// Library/Enumerations/Mode/ProcessingMode
{attribute 'qualified_only'}
// ------------------------------------------------------------------------- 
//  SRCI Robot Library                                                
// ------------------------------------------------------------------------- 
//                                                                           
//  Object:      ProcessingMode                                       
//  Author:      Thorsten Brach                                                
//  Date:        2024-06-01
//
//  Description:                                              
//   
//                                                                           
//  Copyright: 
//    (C) 2024 Thorsten Brach. All rights reserved                                                                                                                                            
//             Licensed under the LGPL-3.0 license.
//                                                                           
//  Disclaimer:                                                                           
//    This project is provided without any guarantee and can be used for   
//    private and commercial purposes. Any use is at the user’s 
//    own risk and responsibility.
//
// -------------------------------------------------------------------------
TYPE ProcessingMode :
(
  /// Command is buffered in sequence buffer and executed once
  BUFFERED := 0,
  /// Command is buffered in sequence buffer, aborts and empties previous commands in sequence buffer, and is executed once
  ABORTING := 1,
  /// Command is buffered in parallel buffer and executed once
  PARALLEL := 2,
  /// Command is buffered in parallel buffer and executed repeatedly until deliberate deactivation by user
  CONTINUOUS := 3,
  /// CMD execution is stopped and/or CMD is removed from the buffer
  DEACTIVATE := 9,
  /// Command is buffered in sequence buffer and executed once (Trigger based)
  TRIGGER_BUFFERED := 10,
  /// Command is buffered in sequence buffer, aborts and empties previous commands in sequence buffer, and is executed once (Trigger based)
  TRIGGER_ABORTING := 11,
  /// Command is buffered in parallel buffer and executed once (Trigger based)
  TRIGGER_ONCE := 12,
  /// Command is buffered in parallel buffer and executed repeatedly until deliberate deactivation by user (Trigger based)
  TRIGGER_CONTINUOUS := 13,
  /// Command is buffered and executed multiple times when triggered. The CMD remains in the buffer until removed by the user.
  TRIGGER_MULTIPLE := 14
)USINT;
END_TYPE

// Library/Enumerations/Mode/ResistanceForceMode
{attribute 'qualified_only'}
// ------------------------------------------------------------------------- 
//  SRCI Robot Library                                                
// ------------------------------------------------------------------------- 
//                                                                           
//  Object:      ResistanceForceMode                                       
//  Author:      Thorsten Brach                                                
//  Date:        2024-06-01
//
//  Description:                                              
//   
//                                                                           
//  Copyright: 
//    (C) 2024 Thorsten Brach. All rights reserved                                                                                                                                            
//             Licensed under the LGPL-3.0 license.
//                                                                           
//  Disclaimer:                                                                           
//    This project is provided without any guarantee and can be used for   
//    private and commercial purposes. Any use is at the user’s 
//    own risk and responsibility.
//
// -------------------------------------------------------------------------
TYPE ResistanceForceMode :
(
  /// 0 (default): ResistanceForceTCP.
  /// Set "0" to set the resistance of the RA against the external force at the TCP.
  RESISTANCE_FORCE_TCP := 0,
  
  /// 1: ResistanceForceAxis.
  /// Set "1" to set the resistance of the RA against the external force for each axis independently.
  RESISTANCE_FORCE_AXIS := 1
)USINT;
END_TYPE

// Library/Enumerations/Mode/ReturnMode
{attribute 'qualified_only'}
TYPE ReturnMode :
(
  /// Interrupt position
  INTERRUPT_POSITION := 0,
  /// End position
  END_POSITION := 1
)BYTE;
END_TYPE

// Library/Enumerations/Mode/SensorConnectionMode
{attribute 'qualified_only'}
// ------------------------------------------------------------------------- 
//  SRCI Robot Library                                                
// ------------------------------------------------------------------------- 
//                                                                           
//  Object:      SensorConnectionMode                                       
//  Author:      Thorsten Brach                                                
//  Date:        2024-06-01
//
//  Description:                                              
//   
//                                                                           
//  Copyright: 
//    (C) 2024 Thorsten Brach. All rights reserved                                                                                                                                            
//             Licensed under the LGPL-3.0 license.
//                                                                           
//  Disclaimer:                                                                           
//    This project is provided without any guarantee and can be used for   
//    private and commercial purposes. Any use is at the user’s 
//    own risk and responsibility.
//
// -------------------------------------------------------------------------
TYPE SensorConnectionMode :
(
  /// RC sensor and algorithm
  /// Force-Torque-Sensor connected to RC
  /// Control algorithm in RC
  RC_SENSOR_ALGORITHM := 0,
  
  /// PLC sensor and RC algorithm
  /// Force-Torque-Sensor connected to PLC
  /// Control algorithm in RC
  PLC_SENSOR_RC_ALGORITHM := 1,
  
  /// PLC sensor and algorithm
  /// Force-Torque-Sensor connected to PLC
  /// Control algorithm in PLC
  PLC_SENSOR_ALGORITHM := 2
)USINT;
END_TYPE

// Library/Enumerations/Mode/SingularityAvoidanceMode
{attribute 'qualified_only'}
// ------------------------------------------------------------------------- 
//  SRCI Robot Library                                                
// ------------------------------------------------------------------------- 
//                                                                           
//  Object:      SingularityAvoidanceMode                                       
//  Author:      Thorsten Brach                                                
//  Date:        2024-06-01
//
//  Description:                                              
//   
//                                                                           
//  Copyright: 
//    (C) 2024 Thorsten Brach. All rights reserved                                                                                                                                            
//             Licensed under the LGPL-3.0 license.
//                                                                           
//  Disclaimer:                                                                           
//    This project is provided without any guarantee and can be used for   
//    private and commercial purposes. Any use is at the user’s 
//    own risk and responsibility.
//
// -------------------------------------------------------------------------
TYPE SingularityAvoidanceMode :
(
  /// 0: NoChange (default)
  /// Allow movement of one or more joints to avoid singularities without a change of the orientation
  NO_CHANGE := 0,
  
  /// 1: Lock J4
  /// Lock the 4th joint to avoid singularities
  LOCK_J4 := 1,
  
  /// 2: ToolOrientation
  /// Allow a small movement of the tool orientation to avoid singularities
  TOOL_ORIENTATION := 2
)USINT;
END_TYPE

// Library/Enumerations/Mode/SplineMode
{attribute 'qualified_only'}
// ------------------------------------------------------------------------- 
//  SRCI Robot Library                                                
// ------------------------------------------------------------------------- 
//                                                                           
//  Object:      SplineMode                                       
//  Author:      Thorsten Brach                                                
//  Date:        2024-06-01
//
//  Description:                                              
//   
//                                                                           
//  Copyright: 
//    (C) 2024 Thorsten Brach. All rights reserved                                                                                                                                            
//             Licensed under the LGPL-3.0 license.
//                                                                           
//  Disclaimer:                                                                           
//    This project is provided without any guarantee and can be used for   
//    private and commercial purposes. Any use is at the user’s 
//    own risk and responsibility.
//
// -------------------------------------------------------------------------
TYPE SplineMode :
(
  /// 0: Discrete Points
  DISCRETE_POINTS := 0,
  /// 1: Bézier Spline
  BEZIER_SPLINE := 1,
  /// 2: B-Splines
  B_SPLINES := 2,
  /// 3: Cubic Hermite Spline
  CUBIC_HERMITE_SPLINE := 3,
  /// 4: C-Splines
  C_SPLINES := 4
)UINT;
END_TYPE

// Library/Enumerations/Mode/StepMode
{attribute 'qualified_only'}
// ------------------------------------------------------------------------- 
//  SRCI Robot Library                                                
// ------------------------------------------------------------------------- 
//                                                                           
//  Object:      StepMode                                       
//  Author:      Thorsten Brach                                                
//  Date:        2024-06-01
//
//  Description:                                              
//   
//                                                                           
//  Copyright: 
//    (C) 2024 Thorsten Brach. All rights reserved                                                                                                                                            
//             Licensed under the LGPL-3.0 license.
//                                                                           
//  Disclaimer:                                                                           
//    This project is provided without any guarantee and can be used for   
//    private and commercial purposes. Any use is at the user’s 
//    own risk and responsibility.
//
// -------------------------------------------------------------------------
TYPE StepMode :
(
  /// StepMode is deactivated
  DEACTIVATE := 0,
  /// Blending
  /// • The robot moves on the blended trajectory
  /// • The movement is interrupted when the active segment changes
  BLENDING := 1,
  ///Exact stop
  /// • The robot moves to the defined target positions without blending
  /// • The movement is interrupted when the defined target position is reached
  EXACT_STOP := 2
)USINT;
END_TYPE

// Library/Enumerations/Mode/StopMode
{attribute 'qualified_only'}
// ------------------------------------------------------------------------- 
//  SRCI Robot Library                                                
// ------------------------------------------------------------------------- 
//                                                                           
//  Object:      StopMode                                       
//  Author:      Thorsten Brach                                                
//  Date:        2024-06-01
//
//  Description:                                              
//   
//                                                                           
//  Copyright: 
//    (C) 2024 Thorsten Brach. All rights reserved                                                                                                                                            
//             Licensed under the LGPL-3.0 license.
//                                                                           
//  Disclaimer:                                                                           
//    This project is provided without any guarantee and can be used for   
//    private and commercial purposes. Any use is at the user’s 
//    own risk and responsibility.
//
// -------------------------------------------------------------------------
TYPE StopMode :
(
  /// 0: Stop via JobID (default)
  /// TargetID is interpreted as JobID
  /// All instances of the defined JobID are stopped
  STOP_JOB_ID := 0,  
  /// 1: Stop via InstanceID
  /// TargetID is interpreted as InstanceID
  /// The instance of the defined InstanceID is stopped
  STOP_INSTANCE_ID := 1,  
  /// 2: Stop all subprograms
  /// All subprograms independent of the input parameter value of TargetID are stopped
  STOP_ALL_SUBPROGRAMS := 2
)USINT;
END_TYPE

// Library/Enumerations/Mode/SyncInMode
{attribute 'qualified_only'}
// ------------------------------------------------------------------------- 
//  SRCI Robot Library                                                
// ------------------------------------------------------------------------- 
//                                                                           
//  Object:      SyncInMode                                       
//  Author:      Thorsten Brach                                                
//  Date:        2024-06-01
//
//  Description:                                              
//   
//                                                                           
//  Copyright: 
//    (C) 2024 Thorsten Brach. All rights reserved                                                                                                                                            
//             Licensed under the LGPL-3.0 license.
//                                                                           
//  Disclaimer:                                                                           
//    This project is provided without any guarantee and can be used for   
//    private and commercial purposes. Any use is at the user’s 
//    own risk and responsibility.
//
// -------------------------------------------------------------------------
TYPE SyncInMode :
(
  /// • When work piece enters "SyncInZone"
  /// • Start synchronization as soon as possible within defined acceleration and velocity limits
  IN_SYNC_IN_ZONE := 0,
  /// • Start synchronization after specific distance after execution
  /// • "SynInZone" ignored
  AFTER_DISTANCE := 1,
  /// • Start synchronization after specific time after execution
  /// • "SynInZone" ignored
  AFTER_TIME := 2,
  /// • As soon as possible within defined acceleration and velocity limits
  /// • "SynInZone" ignored
  IMMEDIATELY := 3
)USINT;
END_TYPE

// Library/Enumerations/Mode/SyncMode
{attribute 'qualified_only'}
// ------------------------------------------------------------------------- 
//  SRCI Robot Library                                                
// ------------------------------------------------------------------------- 
//                                                                           
//  Object:      SyncMode                                       
//  Author:      Thorsten Brach                                                
//  Date:        2024-06-01
//
//  Description:                                              
//   
//                                                                           
//  Copyright: 
//    (C) 2024 Thorsten Brach. All rights reserved                                                                                                                                            
//             Licensed under the LGPL-3.0 license.
//                                                                           
//  Disclaimer:                                                                           
//    This project is provided without any guarantee and can be used for   
//    private and commercial purposes. Any use is at the user’s 
//    own risk and responsibility.
//
// -------------------------------------------------------------------------
TYPE SyncMode :
(
  /// No synchronization will be executed
  NO_SYNCHRONIZATION := 0,
  /// Server data will be overwritten immediately by client data
  CLIENT_TO_SERVER := 1,
  /// Client data will be overwritten immediately by server data
  SERVER_TO_CLIENT := 2,
  /// Server or client data will be overwritten immediately by changed data
  AUTOMATIC := 3
)USINT;
END_TYPE

// Library/Enumerations/Mode/ThresholdMode
{attribute 'qualified_only'}
// ------------------------------------------------------------------------- 
//  SRCI Robot Library                                                
// ------------------------------------------------------------------------- 
//                                                                           
//  Object:      ThresholdMode                                       
//  Author:      Thorsten Brach                                                
//  Date:        2024-06-01
//
//  Description:                                              
//   
//                                                                           
//  Copyright: 
//    (C) 2024 Thorsten Brach. All rights reserved                                                                                                                                            
//             Licensed under the LGPL-3.0 license.
//                                                                           
//  Disclaimer:                                                                           
//    This project is provided without any guarantee and can be used for   
//    private and commercial purposes. Any use is at the user’s 
//    own risk and responsibility.
//
// -------------------------------------------------------------------------
TYPE ThresholdMode :
(
  /// Automatic.
  AUTOMATIC := 0,
  /// Manual (according to LimitAxis)
  MANUAL    := 1
)USINT;
END_TYPE

// Library/Enumerations/Mode/ToolCalculationMode
{attribute 'qualified_only'}
// ------------------------------------------------------------------------- 
//  SRCI Robot Library                                                
// ------------------------------------------------------------------------- 
//                                                                           
//  Object:      ToolCalculationMode                                       
//  Author:      Thorsten Brach                                                
//  Date:        2024-06-01
//
//  Description:                                              
//   
//                                                                           
//  Copyright: 
//    (C) 2024 Thorsten Brach. All rights reserved                                                                                                                                            
//             Licensed under the LGPL-3.0 license.
//                                                                           
//  Disclaimer:                                                                           
//    This project is provided without any guarantee and can be used for   
//    private and commercial purposes. Any use is at the user’s 
//    own risk and responsibility.
//
// -------------------------------------------------------------------------
TYPE ToolCalculationMode :
(
  /// 0: Two Point + Z-Method (default)
  TWO_POINT_Z_METHOD := 0,        
  /// 1: Three-Point-Method
  THREE_POINT_METHOD := 1,        
  /// 2: Four-Point-Method
  FOUR_POINT_METHOD := 2,        
  /// 3: Five-Point-Method
  FIVE_POINT_METHOD := 3,        
  /// 4: Six-Point-Method
  SIX_POINT_METHOD := 4,        
  /// 5: ABC-World-Method
  ABC_WORLD_METHOD := 5,        
  /// 6: ABC-Two-Point-Method
  ABC_TWO_POINT_METHOD := 6
)SINT;
END_TYPE

// Library/Enumerations/Mode/TrajectoryMode
{attribute 'qualified_only'}
// ------------------------------------------------------------------------- 
//  SRCI Robot Library                                                
// ------------------------------------------------------------------------- 
//                                                                           
//  Object:      TrajectoryMode                                       
//  Author:      Thorsten Brach                                                
//  Date:        2024-06-01
//
//  Description:                                              
//   
//                                                                           
//  Copyright: 
//    (C) 2024 Thorsten Brach. All rights reserved                                                                                                                                            
//             Licensed under the LGPL-3.0 license.
//                                                                           
//  Disclaimer:                                                                           
//    This project is provided without any guarantee and can be used for   
//    private and commercial purposes. Any use is at the user’s 
//    own risk and responsibility.
//
// -------------------------------------------------------------------------
TYPE TrajectoryMode :
(
  /// Invalid (default)
  INVALID := 0,
  /// Linear movement
  LINEAR_MOVEMENT := 1,
  /// PTP movement
  PTP_MOVEMENT := 2
)USINT;
END_TYPE

// Library/Enumerations/Mode/TransformMode
{attribute 'qualified_only'}
// ------------------------------------------------------------------------- 
//  SRCI Robot Library                                                
// ------------------------------------------------------------------------- 
//                                                                           
//  Object:      TransformMode                                       
//  Author:      Thorsten Brach                                                
//  Date:        2024-06-01
//
//  Description:                                              
//   
//                                                                           
//  Copyright: 
//    (C) 2024 Thorsten Brach. All rights reserved                                                                                                                                            
//             Licensed under the LGPL-3.0 license.
//                                                                           
//  Disclaimer:                                                                           
//    This project is provided without any guarantee and can be used for   
//    private and commercial purposes. Any use is at the user’s 
//    own risk and responsibility.
//
// -------------------------------------------------------------------------
TYPE TransformMode :
(
  /// 0 (default): Mirror at Point with mirroring of the target position’s orientation
  /// Requires for the mirror Point the "TransformationParameter_1" and the "TransformationParameter_2" set to "Not used"
  MIRROR_AT_POINT := 0,  
  /// 1: Mirror at Straight Line with mirroring of the target position’s orientation
  /// Requires for the Straight Line the "TransformationParameter_1" and the "TransformationParameter_2" set to "X-Axis", "Y-Axis" or "Z-Axis"
  MIRROR_AT_STRAIGHT_LINE := 1,  
  /// 2: Mirror at Plane with mirroring of the target position’s orientation
  /// Requires for the Plane the "TransformationParameter_1" and the "TransformationParameter_2" set to "XY-Axis", "XZ-Axis" or "YZ-Axis"
  MIRROR_AT_PLANE := 2,  
  /// 3: Rotate around Straight Line with rotation of the target position’s orientation
  /// Requires for the Straight Line the "TransformationParameter_1" and the "TransformationParameter_2" set to "X-Axis", "Y-Axis" or "Z-Axis"
  /// Requires for the parameter "RotationAngle"
  ROTATE_AROUND_STRAIGHT_LINE := 3,  
  /// 4: Shift by Vector
  /// Requires for the shifting Vector defined by the Point the "TransformationParameter_1" and the "TransformationParameter_2" set to "Not used"
  /// Requires for the shifting shortest Vector to the Straight Line the "TransformationParameter_1" and the "TransformationParameter_2" set to "X-Axis", "Y-Axis" or "Z-Axis"
  /// Requires for the shifting shortest Vector to the Plane the "TransformationParameter_1" and the "TransformationParameter_2" set to "XY-Axis", "XZ-Axis" or "YZ-Axis"
  SHIFT_BY_VECTOR := 4
)SINT;
END_TYPE

// Library/Enumerations/Mode/TriggerModeIo
{attribute 'qualified_only'}
// ------------------------------------------------------------------------- 
//  SRCI Robot Library                                                
// ------------------------------------------------------------------------- 
//                                                                           
//  Object:      TriggerModeIo                                       
//  Author:      Thorsten Brach                                                
//  Date:        2024-06-01
//
//  Description:                                              
//   
//                                                                           
//  Copyright: 
//    C) 2024 Thorsten Brach. All rights reserved                                                                                                                                            
//             Licensed under the LGPL-3.0 license.
//                                                                           
//  Disclaimer:                                                                           
//    This project is provided without any guarantee and can be used for   
//    private and commercial purposes. Any use is at the user’s 
//    own risk and responsibility.
//
// -------------------------------------------------------------------------
TYPE TriggerModeIo :
(
  /// Invalid (default)
  INVALID := 0,  
  /// Digital Input Rising Edge
  DIGITAL_INPUT_RISING_EDGE := 10,
  /// Digital Input Falling Edge
  DIGITAL_INPUT_FALLING_EDGE := 11,
  /// Digital Input Rising or Falling Edge
  DIGITAL_INPUT_RISING_OR_FALLING_EDGE := 12,
  /// Digital Input Rising or Falling Edge (Inverted)
  DIGITAL_INPUT_RISING_OR_FALLING_EDGE_INVERTED := 13,
  /// Digital Output Rising Edge
  DIGITAL_OUTPUT_RISING_EDGE := 20,
  /// Digital Output Falling Edge
  DIGITAL_OUTPUT_FALLING_EDGE := 21,
  /// Digital Output Rising or Falling Edge
  DIGITAL_OUTPUT_RISING_OR_FALLING_EDGE := 22,
  /// Digital Output Rising or Falling Edge (Inverted)
  DIGITAL_OUTPUT_RISING_OR_FALLING_EDGE_INVERTED := 23,
  /// Analog Input Exceeding Defined Threshold
  ANALOG_INPUT_EXCEEDING_DEFINED_THRESHOLD := 30,
  /// Analog Input Falling Below Defined Threshold
  ANALOG_INPUT_FALLING_BELOW_DEFINED_THRESHOLD := 31,
  /// Analog Input Exceeding or Falling Below Defined Threshold
  ANALOG_INPUT_EXCEEDING_OR_FALLING_BELOW_DEFINED_THRESHOLD := 32,
  /// Analog Input Exceeding or Falling Below Defined Threshold (Inverted)
  ANALOG_INPUT_EXCEEDING_OR_FALLING_BELOW_DEFINED_THRESHOLD_INVERTED := 33,
  /// Analog Input Entering Defined Range
  ANALOG_INPUT_ENTERING_DEFINED_RANGE := 34,
  /// Analog Input Leaving Defined Range
  ANALOG_INPUT_LEAVING_DEFINED_RANGE := 35,
  /// Analog Input Entering or Leaving Defined Range
  ANALOG_INPUT_ENTERING_OR_LEAVING_DEFINED_RANGE := 36,
  /// Analog Input Entering or Leaving Defined Range (Inverted)
  ANALOG_INPUT_ENTERING_OR_LEAVING_DEFINED_RANGE_INVERTED := 37,
  /// Analog Output Exceeding Defined Threshold
  ANALOG_OUTPUT_EXCEEDING_DEFINED_THRESHOLD := 40,
  /// Analog Output Falling Below Defined Threshold
  ANALOG_OUTPUT_FALLING_BELOW_DEFINED_THRESHOLD := 41,
  /// Analog Output Exceeding or Falling Below Defined Threshold
  ANALOG_OUTPUT_EXCEEDING_OR_FALLING_BELOW_DEFINED_THRESHOLD := 42,
  /// Analog Output Exceeding or Falling Below Defined Threshold (Inverted)
  ANALOG_OUTPUT_EXCEEDING_OR_FALLING_BELOW_DEFINED_THRESHOLD_INVERTED := 43,
  /// Analog Output Entering Defined Range
  ANALOG_OUTPUT_ENTERING_DEFINED_RANGE := 44,
  /// Analog Output Leaving Defined Range
  ANALOG_OUTPUT_LEAVING_DEFINED_RANGE := 45,
  /// Analog Output Entering or Leaving Defined Range
  ANALOG_OUTPUT_ENTERING_OR_LEAVING_DEFINED_RANGE := 46,
  /// Analog Output Entering or Leaving Defined Range (Inverted)
  ANALOG_OUTPUT_ENTERING_OR_LEAVING_DEFINED_RANGE_INVERTED := 47,
  /// Integer Register Exceeding Defined Threshold
  INTEGER_REGISTER_EXCEEDING_DEFINED_THRESHOLD := 50,
  /// Integer Register Falling Below Defined Threshold
  INTEGER_REGISTER_FALLING_BELOW_DEFINED_THRESHOLD := 51,
  /// Integer Register Exceeding or Falling Below Defined Threshold
  INTEGER_REGISTER_EXCEEDING_OR_FALLING_BELOW_DEFINED_THRESHOLD := 52,
  /// Integer Register Exceeding or Falling Below Defined Value (Inverted)
  INTEGER_REGISTER_EXCEEDING_OR_FALLING_BELOW_DEFINED_VALUE_INVERTED := 53,
  /// Integer Register Entering Defined Range
  INTEGER_REGISTER_ENTERING_DEFINED_RANGE := 54,
  /// Integer Register Leaving Defined Range
  INTEGER_REGISTER_LEAVING_DEFINED_RANGE := 55,
  /// Integer Register Entering or Leaving Defined Range
  INTEGER_REGISTER_ENTERING_OR_LEAVING_DEFINED_RANGE := 56,
  /// Integer Register Entering or Leaving Defined Range (Inverted)
  INTEGER_REGISTER_ENTERING_OR_LEAVING_DEFINED_RANGE_INVERTED := 57,
  /// Real Register Exceeding Defined Threshold
  REAL_REGISTER_EXCEEDING_DEFINED_THRESHOLD := 60,
  /// Real Register Falling Below Defined Threshold
  REAL_REGISTER_FALLING_BELOW_DEFINED_THRESHOLD := 61,
  /// Real Register Exceeding or Falling Below Defined Threshold
  REAL_REGISTER_EXCEEDING_OR_FALLING_BELOW_DEFINED_THRESHOLD := 62,
  /// Real Register Exceeding or Falling Below Defined Threshold (Inverted)
  REAL_REGISTER_EXCEEDING_OR_FALLING_BELOW_DEFINED_THRESHOLD_INVERTED := 63,
  /// Real Register Entering Defined Range
  REAL_REGISTER_ENTERING_DEFINED_RANGE := 64,
  /// Real Register Leaving Defined Range
  REAL_REGISTER_LEAVING_DEFINED_RANGE := 65,
  /// Real Register Entering or Leaving Defined Range
  REAL_REGISTER_ENTERING_OR_LEAVING_DEFINED_RANGE := 66,
  /// Real Register Entering or Leaving Defined Range (Inverted)
  REAL_REGISTER_ENTERING_OR_LEAVING_DEFINED_RANGE_INVERTED := 67
)SINT;
END_TYPE

// Library/Enumerations/Mode/TriggerModeLimit
{attribute 'qualified_only'}
// ------------------------------------------------------------------------- 
//  SRCI Robot Library                                                
// ------------------------------------------------------------------------- 
//                                                                           
//  Object:      TriggerModeLimit                                       
//  Author:      Thorsten Brach                                                
//  Date:        2024-06-01
//
//  Description:                                              
//   
//                                                                           
//  Copyright: 
//    (C) 2024 Thorsten Brach. All rights reserved                                                                                                                                            
//             Licensed under the LGPL-3.0 license.
//                                                                           
//  Disclaimer:                                                                           
//    This project is provided without any guarantee and can be used for   
//    private and commercial purposes. Any use is at the user’s 
//    own risk and responsibility.
//
// -------------------------------------------------------------------------
TYPE TriggerModeLimit :
(
  /// 0: Invalid (default)
  INVALID := 0,
  /// 1: Joint current in mA
  JOINT_CURRENT := 1,
  /// 2: Force in Nm
  FORCE := 2,
  /// 3: Following error. The distance of the robot position from the path that was calculated
  FOLLOWING_ERROR := 3,
  /// Temperature in °C
  TEMPERATURE := 4  
)SINT;
END_TYPE

// Library/Enumerations/Mode/TriggerModeMeasurement
{attribute 'qualified_only'}
// ------------------------------------------------------------------------- 
//  SRCI Robot Library                                                
// ------------------------------------------------------------------------- 
//                                                                           
//  Object:      TriggerModeMeasurement                                       
//  Author:      Thorsten Brach                                                
//  Date:        2024-06-01
//
//  Description:                                              
//   
//                                                                           
//  Copyright: 
//    (C) 2024 Thorsten Brach. All rights reserved                                                                                                                                            
//             Licensed under the LGPL-3.0 license.
//                                                                           
//  Disclaimer:                                                                           
//    This project is provided without any guarantee and can be used for   
//    private and commercial purposes. Any use is at the user’s 
//    own risk and responsibility.
//
// -------------------------------------------------------------------------
TYPE TriggerModeMeasurement :
(
  /// (default) No trigger related behavior
  NO_TRIGGER := 0,
  /// 1: Starts the measurement with the positive trigger event and stops it with the negative trigger event 
  ///    when the trigger function with the identical EmitterID is activated.
  POSITIVE_START_NEGATIVE_STOP := 1,
  /// 2: Starts and stops the measurement with the positive trigger event 
  ///    when the trigger function with the identical EmitterID is activated.
  POSITIVE_START_STOP := 2
)USINT;
END_TYPE

// Library/Enumerations/Mode/TriggerReactionMode
{attribute 'qualified_only'}
// ------------------------------------------------------------------------- 
//  SRCI Robot Library                                                
// ------------------------------------------------------------------------- 
//                                                                           
//  Object:      TriggerReactionMode                                       
//  Author:      Thorsten Brach                                                
//  Date:        2024-06-01
//
//  Description:                                              
//   
//                                                                           
//  Copyright: 
//    (C) 2024 Thorsten Brach. All rights reserved                                                                                                                                            
//             Licensed under the LGPL-3.0 license.
//                                                                           
//  Disclaimer:                                                                           
//    This project is provided without any guarantee and can be used for   
//    private and commercial purposes. Any use is at the user’s 
//    own risk and responsibility.
//
// -------------------------------------------------------------------------
TYPE TriggerReactionMode :
(
/// No reaction (default).
  NO_REACTION := 0,
  /// Interrupt: Robot movement is paused. Movement can be continued by function GroupContinue.
  INTERRUPT := 1,
  /// GroupStop: Robot stops the movement and brings all axes to a halt. Movements aborted by this command cannot be continued.
  GROUP_STOP := 2,
  /// Disable robot: The robot’s drives are disabled. This leads to the robot state "Not enabled" (see chapter 5.5.3).
  DISABLE_ROBOT := 3,
  /// Stop actual motion command: Robot movement is paused. Movement can be continued by the next motion command.
  STOP_ACTUAL_MOTION_COMMAND := 4
)SINT;
END_TYPE

// Library/Enumerations/Mode/TurnMode
{attribute 'qualified_only'}
// ------------------------------------------------------------------------- 
//  SRCI Robot Library                                                
// ------------------------------------------------------------------------- 
//                                                                           
//  Object:      TurnMode                                       
//  Author:      Thorsten Brach                                                
//  Date:        2024-06-01
//
//  Description:                                              
//   
//                                                                           
//  Copyright: 
//    (C) 2024 Thorsten Brach. All rights reserved                                                                                                                                            
//             Licensed under the LGPL-3.0 license.
//                                                                           
//  Disclaimer:                                                                           
//    This project is provided without any guarantee and can be used for   
//    private and commercial purposes. Any use is at the user’s 
//    own risk and responsibility.
//
// -------------------------------------------------------------------------
TYPE TurnMode :
(
  /// Use TurnNumber in position
  USE_TURN_NUMBER := 0,
  ///  Do not change TurnNumber with this movement
  SAME            := 1,
  /// TurnNumber in position is not used but the Robot is free to change TurnNumber
  FREE            := 2
)USINT;
END_TYPE

// Library/Enumerations/Mode/WorkAreaReactionMode
{attribute 'qualified_only'}
// ------------------------------------------------------------------------- 
//  SRCI Robot Library                                                
// ------------------------------------------------------------------------- 
//                                                                           
//  Object:      WorkAreaReactionMode                                       
//  Author:      Thorsten Brach                                                
//  Date:        2024-06-01
//
//  Description:                                              
//   
//                                                                           
//  Copyright: 
//    (C) 2024 Thorsten Brach. All rights reserved                                                                                                                                            
//             Licensed under the LGPL-3.0 license.
//                                                                           
//  Disclaimer:                                                                           
//    This project is provided without any guarantee and can be used for   
//    private and commercial purposes. Any use is at the user’s 
//    own risk and responsibility.
//
// -------------------------------------------------------------------------
TYPE WorkAreaReactionMode :
(
  /// 0: No reaction (default)
  /// • RC reports violation
  /// • Robot is not stopped
  NO_REACTION := 0,
  /// 
  /// 1: Abort
  /// • RC reports violation
  /// • RC returns error
  /// • Robot is stopped
  /// • Sequence buffer emptied
  ABORT := 1,
  /// 2: Interrupt
  /// • RC reports violation
  /// • Robot movement is paused
  /// • Movement can be continued by function GroupContinue
   INTERRUPT := 2
)USINT;
END_TYPE

// Library/Enumerations/State/ActiveCommandRegisterState
{attribute 'qualified_only'}
// ------------------------------------------------------------------------- 
//  SRCI Robot Library                                                
// ------------------------------------------------------------------------- 
//                                                                           
//  Object:      ActiveCommandRegisterState                                       
//  Author:      Thorsten Brach                                                
//  Date:        2024-06-01
//
//  Description:                                              
//   
//                                                                           
//  Copyright: 
//    (C) 2024 Thorsten Brach. All rights reserved                                                                                                                                            
//             Licensed under the LGPL-3.0 license.
//                                                                           
//  Disclaimer:                                                                           
//    This project is provided without any guarantee and can be used for   
//    private and commercial purposes. Any use is at the user’s 
//    own risk and responsibility.
//
// -------------------------------------------------------------------------
TYPE ActiveCommandRegisterState :
(
  /// IS_FREE denotes not used but available resources (empty slots in the ACR).
  IS_FREE        := 0,
  /// IS_PROCESSING CMDs are actively being processed by client or server. 
  /// In terms of CMD category, IS_PROCESSING also describes commands whose tasks are not currently being executed (not ACTIVE), 
  /// but e.g. a CMD waiting in the Sequence buffer.
  IS_PROCESSING := 1,
  /// IS_FINAL states are reached on CMD termination. Execution of this Task has been finished and its results can be examined.
  IS_FINAL    := 2
);
END_TYPE

// Library/Enumerations/State/BufferStateCmd
{attribute 'qualified_only'}
// ------------------------------------------------------------------------- 
//  SRCI Robot Library                                                
// ------------------------------------------------------------------------- 
//                                                                           
//  Object:      BufferStateCmd                                       
//  Author:      Thorsten Brach                                                
//  Date:        2024-06-01
//
//  Description:                                              
//   
//                                                                           
//  Copyright: 
//    (C) 2024 Thorsten Brach. All rights reserved                                                                                                                                            
//             Licensed under the LGPL-3.0 license.
//                                                                           
//  Disclaimer:                                                                           
//    This project is provided without any guarantee and can be used for   
//    private and commercial purposes. Any use is at the user’s 
//    own risk and responsibility.
//
// -------------------------------------------------------------------------
TYPE BufferStateCmd :
(
 // PDF Page 353 
  EMPTY            := 0,
  CREATED          := 1,
  UPDATE_AVAILABLE := 2,
  SENDING          := 3,
  PROCESSED        := 4  
);
END_TYPE

// Library/Enumerations/State/BufferStateRsp
{attribute 'qualified_only'}
// ------------------------------------------------------------------------- 
//  SRCI Robot Library                                                
// ------------------------------------------------------------------------- 
//                                                                           
//  Object:      BufferStateRsp                                       
//  Author:      Thorsten Brach                                                
//  Date:        2024-06-01
//
//  Description:                                              
//   
//                                                                           
//  Copyright: 
//    (C) 2024 Thorsten Brach. All rights reserved                                                                                                                                            
//             Licensed under the LGPL-3.0 license.
//                                                                           
//  Disclaimer:                                                                           
//    This project is provided without any guarantee and can be used for   
//    private and commercial purposes. Any use is at the user’s 
//    own risk and responsibility.
//
// -------------------------------------------------------------------------
TYPE BufferStateRsp :
(
 // PDF Seite 353 
  EMPTY            := 0,
  RECEIVING        := 1,
  RECEIVED         := 2,
  PROCESSED        := 3  
);
END_TYPE

// Library/Enumerations/State/CmdMessageState
{attribute 'qualified_only'}
// ------------------------------------------------------------------------- 
//  SRCI Robot Library                                                
// ------------------------------------------------------------------------- 
//                                                                           
//  Object:      CmdMessageState                                       
//  Author:      Thorsten Brach                                                
//  Date:        2024-06-01
//
//  Description:                                              
//   
//                                                                           
//  Copyright: 
//    (C) 2024 Thorsten Brach. All rights reserved                                                                                                                                            
//             Licensed under the LGPL-3.0 license.
//                                                                           
//  Disclaimer:                                                                           
//    This project is provided without any guarantee and can be used for   
//    private and commercial purposes. Any use is at the user’s 
//    own risk and responsibility.
//
// -------------------------------------------------------------------------
TYPE CmdMessageState :
(
  /// No operation or process is active
  EMPTY := 0,
  /// Created but not yet started
  CREATED := 1,
  /// Buffered and awaiting execution
  BUFFERED := 2,
  /// Buffered in planner for future execution
  BUFFERED_IN_PLANNER := 3,
  /// Currently active and in progress
  ACTIVE := 4,
  /// Interrupted and awaiting continuation
  INTERRUPTED := 5,
  /// Requested for abort
  ABORT_REQUEST := 6,
  /// Successfully completed
  DONE := 10,
  /// Aborted before completion
  ABORTED := 14,
  /// Encountered an error during execution
  ERROR := 15
)USINT;
END_TYPE

// Library/Enumerations/State/FsmState
/// finite state machine
{attribute 'qualified_only'}
TYPE FsmState :
(
  /// READY
  READY := 0,
  /// START
  START,
  /// RUNNING
  RUNNING,
  /// DONE
  DONE,
  /// CANCEL
  CANCEL,
  /// ERROR
  ERROR,
  /// ERROR_CLEAR
  ERROR_CLEAR
);
END_TYPE

// Library/Enumerations/State/InitializationState
{attribute 'qualified_only'}
// ------------------------------------------------------------------------- 
//  SRCI Robot Library                                                
// ------------------------------------------------------------------------- 
//                                                                           
//  Object:      InitializationState                                       
//  Author:      Thorsten Brach                                                
//  Date:        2024-06-01
//
//  Description:                                              
//   
//                                                                           
//  Copyright: 
//    (C) 2024 Thorsten Brach. All rights reserved                                                                                                                                            
//             Licensed under the LGPL-3.0 license.
//                                                                           
//  Disclaimer:                                                                           
//    This project is provided without any guarantee and can be used for   
//    private and commercial purposes. Any use is at the user’s 
//    own risk and responsibility.
//
// -------------------------------------------------------------------------
TYPE InitializationState :
(
  /// Default
  DEFAULT := 0,
  /// Error: Telegram control does not match the telegram state
  ERROR_TELEGRAM_CONTROL := 161,
  /// Error: Initialization lost for unknown reason. See message log after reinitializing
  ERROR_INIT_LOST := 162,
  /// Error: Telegram length does not match the length provided in the communication interface.
  ERROR_TELEGRAM_LENGTH := 163,
  /// Error: Incompatible major SRCI version
  ERROR_INCOMPATIBLE_SRCI := 164,
  /// Error: Lifesign timeout
  ERROR_LIFESIGN_TIMEOUT := 165,
  /// Error: The selected optional cyclic data does not fit in the given telegram size
  ERROR_CYCLIC_DATA_MISMATCH := 166,
  /// Error: The robot interface was reset after being initialized
  ERROR_INTERFACE_RESET := 167,
  /// Error: Telegram sequence timeout
  ERROR_SEQUENCE_TIMEOUT := 168,
  /// Error: The telegram number changed after initialization
  ERROR_TELEGRAM_NUMBER_CHANGED := 169,
  /// Error: Invalid AxesGroupID
  ERROR_INVALID_AXES_GROUP := 170,
  /// Error: Telegram number is invalid. E.g. TwoSequences is only activated in one direction
  ERROR_INVALID_TELEGRAM_NUMBER := 171,
  /// Error: Telegram Number is not supported
  ERROR_TELEGRAM_NUMBER_NOT_SUPPORTED := 172,
  /// Ready to resume: The RC is currently not initialized but has state in the ACR
  READY_TO_RESUME := 253,
  /// Ready for initialization: The RC is currently not initialized and has no state in the ACR
  READY_FOR_INITIALIZATION := 254,
  /// Initialized: The RC state is Initialized
  INITIALIZED := 255
);
END_TYPE

// Library/Enumerations/State/RaPowerState
{attribute 'qualified_only'}
// ------------------------------------------------------------------------- 
//  SRCI Robot Library                                                
// ------------------------------------------------------------------------- 
//                                                                           
//  Object:      RaPowerState                                       
//  Author:      Thorsten Brach                                                
//  Date:        2024-06-01
//
//  Description:                                              
//   
//                                                                           
//  Copyright: 
//    (C) 2024 Thorsten Brach. All rights reserved                                                                                                                                            
//             Licensed under the LGPL-3.0 license.
//                                                                           
//  Disclaimer:                                                                           
//    This project is provided without any guarantee and can be used for   
//    private and commercial purposes. Any use is at the user’s 
//    own risk and responsibility.
//
// -------------------------------------------------------------------------
TYPE RaPowerState :
(
  /// Robot drives disabled. Robot cannot be moved
  NOT_ENABLED := 0,
  /// Robot drives powered on. Robot can be moved according to sequence state
  ENABLED := 1
)USINT;
END_TYPE

// Library/Enumerations/State/RaSequenceState
{attribute 'qualified_only'}
// ------------------------------------------------------------------------- 
//  SRCI Robot Library                                                
// ------------------------------------------------------------------------- 
//                                                                           
//  Object:      RaSequenceState                                       
//  Author:      Thorsten Brach                                                
//  Date:        2024-06-01
//
//  Description:                                              
//   
//                                                                           
//  Copyright: 
//    (C) 2024 Thorsten Brach. All rights reserved                                                                                                                                            
//             Licensed under the LGPL-3.0 license.
//                                                                           
//  Disclaimer:                                                                           
//    This project is provided without any guarantee and can be used for   
//    private and commercial purposes. Any use is at the user’s 
//    own risk and responsibility.
//
// -------------------------------------------------------------------------
TYPE RaSequenceState :
(
  /// Robot can be moved by incoming command
  IDLE := 0,
  /// RC is processing command in active sequence
  EXECUTING := 1,
  /// Interrupt is active. Robot is waiting for Continue
  INTERRUPTED := 2
)USINT;
END_TYPE

// Library/Enumerations/State/RiState
{attribute 'qualified_only'}
// ------------------------------------------------------------------------- 
//  SRCI Robot Library                                                
// ------------------------------------------------------------------------- 
//                                                                           
//  Object:      RiState                                       
//  Author:      Thorsten Brach                                                
//  Date:        2024-06-01
//
//  Description:                                              
//   
//                                                                           
//  Copyright: 
//    (C) 2024 Thorsten Brach. All rights reserved                                                                                                                                            
//             Licensed under the LGPL-3.0 license.
//                                                                           
//  Disclaimer:                                                                           
//    This project is provided without any guarantee and can be used for   
//    private and commercial purposes. Any use is at the user’s 
//    own risk and responsibility.
//
// -------------------------------------------------------------------------
TYPE RiState :
(
  /// RI is not initialized
  NOT_INITIALIZED := 0,
  /// Initialization finished successfully
  INITIALIZED := 1,
  /// Data between RC and PLC has been synchronized
  SYNCHRONIZED := 2
)USINT;
END_TYPE

// Library/Enumerations/State/TelegramState
{attribute 'qualified_only'}
TYPE TelegramState :
(
  /// Default
  UNDEFINED := 0,
  /// Telegram control does not match the telegram state
  ERROR_161 := 161,
  /// Initialization lost for unknown reason. See message log after reinitializing
  ERROR_162 := 162,
  /// Telegram length does not match the length provided in the communication interface.
  ERROR_163 := 163,
  /// Incompatible major SRCI version
  ERROR_164 := 164,
  /// Lifesign timeout
  ERROR_165 := 165,
  /// The selected optional cyclic data does not fit in the given telegram size
  ERROR_166 := 166,
  /// The robot interface was reset after being initialized
  ERROR_167 := 167,
  /// Telegram sequence timeout
  ERROR_168 := 168,
  /// The telegram number changed after initialization
  ERROR_169 := 169,
  /// Invalid AxesGroupID
  ERROR_170 := 170,
  /// Telegram number is invalid. E.g. TwoSequences is only activated in one direction
  ERROR_171 := 171,
  /// Telegram Number is not supported
  ERROR_172 := 172,
  /// The RC is currently not initialized but has state in the ACR
  READY_TO_RESUME := 253,
  /// The RC is currently not initialized and has no state in the ACR
  READY_FOR_INITIALIZATION := 254,
  /// The RC state is Initialized
  INITIALIZED := 255  
)USINT;
END_TYPE

// Library/Enumerations/Type/AreaType
{attribute 'qualified_only'}
// ------------------------------------------------------------------------- 
//  SRCI Robot Library                                                
// ------------------------------------------------------------------------- 
//                                                                           
//  Object:      AreaType                                       
//  Author:      Thorsten Brach                                                
//  Date:        2024-06-01
//
//  Description:                                              
//   
//                                                                           
//  Copyright: 
//    (C) 2024 Thorsten Brach. All rights reserved                                                                                                                                            
//             Licensed under the LGPL-3.0 license.
//                                                                           
//  Disclaimer:                                                                           
//    This project is provided without any guarantee and can be used for   
//    private and commercial purposes. Any use is at the user’s 
//    own risk and responsibility.
//
// -------------------------------------------------------------------------
TYPE AreaType :
(
  /// 0: Axes
  AXES := 0,
  /// 1: Box (default)
  BOX := 1,
  /// 2: Cylinder
  CYLINDER := 2,
  /// 3: Sphere (only DefinitionMode 1)
  SPHERE := 3
)USINT;
END_TYPE

// Library/Enumerations/Type/AxesGroupParameterCmdEntries
{attribute 'qualified_only'}
// ------------------------------------------------------------------------- 
//  SRCI Robot Library                                                
// ------------------------------------------------------------------------- 
//                                                                           
//  Object:      AxesGroupParameterCmdEntries                                       
//  Author:      Thorsten Brach                                                
//  Date:        2024-06-01
//
//  Description:                                              
//   
//                                                                           
//  Copyright: 
//    (C) 2024 Thorsten Brach. All rights reserved                                                                                                                                            
//             Licensed under the LGPL-3.0 license.
//                                                                           
//  Disclaimer:                                                                           
//    This project is provided without any guarantee and can be used for   
//    private and commercial purposes. Any use is at the user’s 
//    own risk and responsibility.
//
// -------------------------------------------------------------------------
TYPE AxesGroupParameterCmdEntries :
(
  /// Handles multiple mechanisms required for operation of the interface
  RobotTask := 0, // No function code  
  /// Read robot-specific data from the RC
  ReadRobotData := 9002,  
  /// Enable/Disable robot into RA power state "Enabled"
  EnableRobot := 1,  
  /// Acknowledgement all pending errors
  GroupReset := 2,  
  /// Read the actual position – TCP: X…RZ + config/Turn, Joint: (J1…E6)
  ReadActualPosition := 3,
  /// Read the actual position cyclically
  ReadActualPositionCyclic := 4,   
  /// Read D-H-parameters of robot
  ReadDHParameter := 5,  
  /// Restart/reboot of the RC
  RestartController := 6,  
  /// Read actual TCP velocity
  ReadActualTCPVelocity := 7,  
  /// Login on RC from PLC
  UserLogin := 8,  
  /// Switch language of robot teach pendant from PLC
  SwitchLanguage := 9,  
  /// Reads and writes specific configuration parameters on RC that are required for the RI to work
  ExchangeConfiguration := 10,  
  /// Set active sequence
  SetSequence := 11,  
  /// Change actual speed override
  ChangeSpeedOverride := 12,  
  /// Read error codes of pending errors and move them into user data block "RobotData"
  ReadMessages := 13,  
  /// Read reference values of robot dynamics for path movement
  ReadRobotReferenceDynamics := 14,  
  /// Change configuration of selected user frame number
  WriteFrameData := 15,  
  /// Change configuration of selected tool number
  WriteToolData := 16,  
  /// Change configuration of selected payload number
  WriteLoadData := 17,  
  /// Write reference values of robot dynamics for path movement
  WriteRobotReferenceDynamics := 18,  
  /// Write default values of dynamic parameters used by move commands
  WriteRobotDefaultDynamics := 19,  
  /// Read default values of dynamic parameters used by move commands
  ReadRobotDefaultDynamics := 20,  
  /// Read content of selected user frame number
  ReadFrameData := 21,  
  /// Read content of selected tool number
  ReadToolData := 22,  
  /// Read content of selected payload number
  ReadLoadData := 23,  
  /// Read actual software limits of the axes Positive and negative Limit of Joint J1…J6, E1…E6
  ReadRobotSWLimits := 24,  
  /// Change robot limits of robot axes (degree)
  WriteRobotSWLimits := 25,  
  /// Switch operation mode of RC (Automatic External, T1 External, T2 External)
  SetOperationMode := 26,  
  /// Read configuration of defined work areas
  ReadWorkArea := 27,  
  /// Define work area
  WriteWorkArea := 28,  
  /// Enable/Disable work areas of RC and check if TCP is inside/outside of active work area
  ActivateWorkArea := 29,  
  /// Monitor enabled work areas
  MonitorWorkArea := 30,  
  /// Jog robot manually
  GroupJog := 31,  
  /// Move the TCP to an absolute cartesian position (linear interpolation)
  MoveLinearAbsolute := 32,  
  /// Move Joints to an absolute cartesian position (Absolute cartesian PTP) (Joint interpolated movement)
  MoveDirectAbsolute := 33,  
  /// Move all joints to an absolute joint position (Absolute Joint PTP)
  MoveAxesAbsolute := 34,  
  /// Abort actual movement and delete buffer
  GroupStop := 35,  
  /// Interrupt active movement, possible to continue movement
  GroupInterrupt := 36,  
  /// Continue interrupted path
  GroupContinue := 37,  
  /// Move the TCP relative to the actual cartesian position (linear interpolation)
  MoveLinearRelative := 38,  
  /// Move Joints relative to relative cartesian position (Relative cartesian PTP) (Joint interpolated movement)
  MoveDirectRelative := 39,  
  /// Move all joints relative to actual joint position (Relative Joint PTP)
  MoveAxesRelative := 40,  
  /// Return to path left during active interrupt
  ReturnToPrimary := 41,  
  /// Move the TCP to an absolute joint position (linear interpolation)
  MoveCircularAbsolute := 42,  
  /// Move the TCP relative to the actual cartesian position (circular interpolation)
  MoveCircularRelative := 43,  
  /// Move the TCP relative to a reference cartesian position (linear interpolation)
  MoveLinearOffset := 44,  
  /// Move the TCP relative to a reference cartesian position (PTPT interpolation)
  MoveDirectOffset := 45,  
  /// Set wait command between motion commands
  WaitTime := 46,  
  /// Linear Move to target position through auxiliary position defined by offset in all dimensions (movement to target position linear)
  MoveApproachLinear := 47,  
  /// Linear Move from actual position to destination through auxiliary position defined by offset in all dimensions (movement to target position linear)
  MoveDepartLinear := 48,  
  /// Direct Move to target position through auxiliary position defined by offset in all dimensions (movement to target posi tion PTP)
  MoveApproachDirect := 49,  
  /// Direct Move from actual position to destination through auxiliary position defined by offset in all dimensions (movement to the target position PTP)
  MoveDepartDirect := 50,  
  /// Move robot into contact with obstruction (mechanical Limit) and hold it in this position
  SearchHardstop := 51,  
  /// Move robot into contact with obstruction (mechanical Limit) and hold it in this position
  SearchHardstopJ := 52,  
  /// Command several interpolated movement of robot arm on linear paths from actual position
  MovePickPlaceLinear := 53,  
  /// Commands interpolated movement of robot arm on a partly undefined path from actual position
  MovePickPlaceDirect := 54,  
  /// Activate conveyor tracking mode
  ActivateConveyorTracking := 55,  
  /// Redefine tracking position for conveyor tracking
  RedefineTrackingPos := 56,  
  /// Synchronize robot with conveyor
  SyncToConveyor := 57,  
  /// Configure conveyor parameters
  ConfigureConveyor := 58,  
  /// Activate superimposed motion of TCP to defined motion
  MoveSuperImposed := 59,  
  /// Activate superimposed motion of TCP to defined motion
  MoveSuperImposedDynamic := 60,  
  /// Read digital input and output group of RC
  ReadDigitalInputs := 61,  
  /// Read digital output group of RC
  ReadDigitalOutputs := 62,  
  /// Write digital output group of RC
  WriteDigitalOutputs := 63,  
  /// Read integer values on RC
  ReadIntegers := 64,  
  /// Read real values on RC
  ReadReals := 65,  
  /// Write integer values on RC
  WriteIntegers := 66,  
  /// Write real values on RC
  WriteReals := 67,  
  /// Set trigger in defined position of path (L = Linear Path) (cartesian) switch periphery.
  MoveLinearCam := 68,  
  /// Set a trigger in a defined position of a path. (PTP)
  MoveDirectCam := 69,  
  /// Set a trigger in a defined position of a circular path
  MoveCircularCam := 70,  
  /// Read analog input of RC
  ReadAnalogInput := 71,  
  /// Read analog output of RC
  ReadAnalogOutput := 72,  
  /// Write analog output of RC
  WriteAnalogOutput := 73,  
  /// Capture trigger Position, measuring input
  MeasuringInput := 74,  
  /// Abort triggering of Position, measuring input
  AbortMeasuringInput := 75,  
  /// Trigger "Actions" based on I/O related events (e.g. change of DI’s state)
  SetTriggerRegister := 76,  
  /// Trigger "Actions" based on physical events (e.g. force limit reached)
  SetTriggerLimit := 77,  
  /// Trigger "Actions" based on physical events (e.g. force limit reached)
  SetTriggerUser := 78,  
  /// Trigger "Actions" based on incoming error event
  SetTriggerError := 79,  
  /// "Action" that initiates specified events when triggered
  ReactAtTrigger := 80,  
  /// Wait to process next command in sequence until trigger signal is received
  WaitForTrigger := 81,  
  /// Read specific parameter of the robot
  ReadSystemVariable := 82,  
  /// Change value of specific vendor parameter
  WriteSystemVariable := 83,  
  /// Calculate Forward Kinematic
  CalculateForwardKinematic := 84,  
  /// Calculate Inverse Kinematic
  CalculateInverseKinematic := 85,  
  /// Calculate cartesian position from existing cartesian position
  CalculateCartesianPosition := 86,  
  /// Calculate tool (TCP) with four-point method
  CalculateTool := 87,  
  /// Calculate frame with three-point method
  CalculateFrame := 88,  
  /// Cancel currently active move command and continue with the next buffered command
  ActivateNextCommand := 89,  
  /// Transform a defined position in space
  ShiftPosition := 90,  
  /// Trigger an action based on a motion-related parameter (e.g. progress of trajectory)
  SetTriggerMotion := 91,  
  /// Release robot arm’s brakes
  OpenBrake := 92,  
  /// Call subprogram stored in RC from PLC
  CallSubprogram := 93,  
  /// Writes cyclic data of called subprogram
  WriteCallSubprogramCyclic := 94,
  /// Reads cyclic data of called subprogram
  ReadCallSubprogramCyclic := 95,
  /// Stops an active subprogram
  StopSubprogram := 96,  
  /// Switch path mode between high and low accuracy
  PathAccuracyMode := 97,  
  /// Activate/Deactivate functionality to avoid singularities
  AvoidSingularity := 98,  
  /// Enables the RC to apply user-defined force/torque through RA’s TCP movement
  ForceControl := 99,  
  /// Commands specified reaction from RA when defined force/torque detected
  ForceLimit := 100,  
  /// Read actual force/torque at TCP
  ReadActualForce := 101,  
  /// Activate robot cycle brake test and give feedback to PLC
  BrakeTest := 102,  
  /// Push robot: Robot calculates opposite vector and moves slowly in that direction
  SoftSwitchTCP := 103,  
  /// Create spline on RC from positions stored in PLC
  CreateSpline := 104,  
  /// Delete spline previously created on RC
  DeleteSpline := 105,  
  /// Move spline previously created on RC
  MoveSpline := 106,  
  /// Create and move spline on RC simultaneously
  DynamicSpline := 107,  
  /// Automatic detection of load data
  LoadMeasurementAutomatic := 108,  
  /// Sequential detection of load data
  LoadMeasurementSequential := 109,  
  /// Turn on/off the collision detection
  CollisionDetection := 110,  
  /// Move the robot axes by hand
  FreeDrive := 111,  
  /// Measure the length of objects in the cartesian space, execution time for specified section of a job or signal output time of a specified signal
  UnitMeasurement := 112,
  /// Maximum entry
  MAX_ENTRY := 113   
)UINT;
END_TYPE

// Library/Enumerations/Type/CmdType
{attribute 'qualified_only'}
// ------------------------------------------------------------------------- 
//  SRCI Robot Library                                                
// ------------------------------------------------------------------------- 
//                                                                           
//  Object:      CmdType                                       
//  Author:      Thorsten Brach                                                
//  Date:        2024-06-01
//
//  Description:                                              
//   
//                                                                           
//  Copyright: 
//    (C) 2024 Thorsten Brach. All rights reserved                                                                                                                                            
//             Licensed under the LGPL-3.0 license.
//                                                                           
//  Disclaimer:                                                                           
//    This project is provided without any guarantee and can be used for   
//    private and commercial purposes. Any use is at the user’s 
//    own risk and responsibility.
//
// -------------------------------------------------------------------------
TYPE CmdType :
(
  /// Handles multiple mechanisms required for operation of the interface
  RobotTask := 0, // No function code  
  /// Read robot-specific data from the RC
  ReadRobotData := 9002,  
  /// Enable/Disable robot into RA power state "Enabled"
  EnableRobot := 1000,  
  /// Acknowledgement all pending errors
  GroupReset := 1001,  
  /// Read the actual position – TCP: X…RZ + config/Turn, Joint: (J1…E6)
  ReadActualPosition := 5100,
  /// Read the actual position cyclically
  ReadActualPositionCyclic := 1, // No function code  
  /// Read D-H-parameters of robot
  ReadDHParameter := 5101,  
  /// Restart/reboot of the RC
  RestartController := 1101,  
  /// Read actual TCP velocity
  ReadActualTCPVelocity := 5111,  
  /// Login on RC from PLC
  UserLogin := 1006,  
  /// Switch language of robot teach pendant from PLC
  SwitchLanguage := 1005,  
  /// Reads and writes specific configuration parameters on RC that are required for the RI to work
  ExchangeConfiguration := 9000,  
  /// Set active sequence
  SetSequence := 1004,  
  /// Change actual speed override
  ChangeSpeedOverride := 2000,  
  /// Read error codes of pending errors and move them into user data block "RobotData"
  ReadMessages := 9001,  
  /// Read reference values of robot dynamics for path movement
  ReadRobotReferenceDynamics := 5105,  
  /// Change configuration of selected user frame number
  WriteFrameData := 5200,  
  /// Change configuration of selected tool number
  WriteToolData := 5205,  
  /// Change configuration of selected payload number
  WriteLoadData := 5201,  
  /// Write reference values of robot dynamics for path movement
  WriteRobotReferenceDynamics := 5203,  
  /// Write default values of dynamic parameters used by move commands
  WriteRobotDefaultDynamics := 5202,  
  /// Read default values of dynamic parameters used by move commands
  ReadRobotDefaultDynamics := 5104,  
  /// Read content of selected user frame number
  ReadFrameData := 5102,  
  /// Read content of selected tool number
  ReadToolData := 5107,  
  /// Read content of selected payload number
  ReadLoadData := 5103,  
  /// Read actual software limits of the axes Positive and negative Limit of Joint J1…J6, E1…E6
  ReadRobotSWLimits := 5106,  
  /// Change robot limits of robot axes (degree)
  WriteRobotSWLimits := 5204,  
  /// Switch operation mode of RC (Automatic External, T1 External, T2 External)
  SetOperationMode := 1003,  
  /// Read configuration of defined work areas
  ReadWorkArea := 7502,  
  /// Define work area
  WriteWorkArea := 7503,  
  /// Enable/Disable work areas of RC and check if TCP is inside/outside of active work area
  ActivateWorkArea := 7500,  
  /// Monitor enabled work areas
  MonitorWorkArea := 7501,  
  /// Jog robot manually
  GroupJog := 2100,  
  /// Move the TCP to an absolute cartesian position (linear interpolation)
  MoveLinearAbsolute := 2103,  
  /// Move Joints to an absolute cartesian position (Absolute cartesian PTP) (Joint interpolated movement)
  MoveDirectAbsolute := 2102,  
  /// Move all joints to an absolute joint position (Absolute Joint PTP)
  MoveAxesAbsolute := 2101,  
  /// Abort actual movement and delete buffer
  GroupStop := 2003,  
  /// Interrupt active movement, possible to continue movement
  GroupInterrupt := 2002,  
  /// Continue interrupted path
  GroupContinue := 2001,  
  /// Move the TCP relative to the actual cartesian position (linear interpolation)
  MoveLinearRelative := 2110,  
  /// Move Joints relative to relative cartesian position (Relative cartesian PTP) (Joint interpolated movement)
  MoveDirectRelative := 2108,  
  /// Move all joints relative to actual joint position (Relative Joint PTP)
  MoveAxesRelative := 2105,  
  /// Return to path left during active interrupt
  ReturnToPrimary := 2104,  
  /// Move the TCP to an absolute joint position (linear interpolation)
  MoveCircularAbsolute := 2109,  
  /// Move the TCP relative to the actual cartesian position (circular interpolation)
  MoveCircularRelative := 2106,  
  /// Move the TCP relative to a reference cartesian position (linear interpolation)
  MoveLinearOffset := 2112,  
  /// Move the TCP relative to a reference cartesian position (PTPT interpolation)
  MoveDirectOffset := 2111,  
  /// Set wait command between motion commands
  WaitTime := 7005,  
  /// Linear Move to target position through auxiliary position defined by offset in all dimensions (movement to target position linear)
  MoveApproachLinear := 2201,  
  /// Linear Move from actual position to destination through auxiliary position defined by offset in all dimensions (movement to target position linear)
  MoveDepartLinear := 2203,  
  /// Direct Move to target position through auxiliary position defined by offset in all dimensions (movement to target posi tion PTP)
  MoveApproachDirect := 2200,  
  /// Direct Move from actual position to destination through auxiliary position defined by offset in all dimensions (movement to the target position PTP)
  MoveDepartDirect := 2202,  
  /// Move robot into contact with obstruction (mechanical Limit) and hold it in this position
  SearchHardstop := 2500,  
  /// Move robot into contact with obstruction (mechanical Limit) and hold it in this position
  SearchHardstopJ := 2501,  
  /// Command several interpolated movement of robot arm on linear paths from actual position
  MovePickPlaceLinear := 2205,  
  /// Commands interpolated movement of robot arm on a partly undefined path from actual position
  MovePickPlaceDirect := 2204,  
  /// Activate conveyor tracking mode
  ActivateConveyorTracking := 2300,  
  /// Redefine tracking position for conveyor tracking
  RedefineTrackingPos := 2302,  
  /// Synchronize robot with conveyor
  SyncToConveyor := 2303,  
  /// Configure conveyor parameters
  ConfigureConveyor := 2301,  
  /// Activate superimposed motion of TCP to defined motion
  MoveSuperImposed := 2502,  
  /// Activate superimposed motion of TCP to defined motion
  MoveSuperImposedDynamic := 2503,  
  /// Read digital input and output group of RC
  ReadDigitalInputs := 6100,  
  /// Read digital output group of RC
  ReadDigitalOutputs := 6101,  
  /// Write digital output group of RC
  WriteDigitalOutputs := 6104,  
  /// Read integer values on RC
  ReadIntegers := 6102,  
  /// Read real values on RC
  ReadReals := 6103,  
  /// Write integer values on RC
  WriteIntegers := 6105,  
  /// Write real values on RC
  WriteReals := 6106,  
  /// Set trigger in defined position of path (L = Linear Path) (cartesian) switch periphery.
  MoveLinearCam := 2402,  
  /// Set a trigger in a defined position of a path. (PTP)
  MoveDirectCam := 2401,  
  /// Set a trigger in a defined position of a circular path
  MoveCircularCam := 2400,  
  /// Read analog input of RC
  ReadAnalogInput := 6107,  
  /// Read analog output of RC
  ReadAnalogOutput := 6108,  
  /// Write analog output of RC
  WriteAnalogOutput := 6109,  
  /// Capture trigger Position, measuring input
  MeasuringInput := 6001,  
  /// Abort triggering of Position, measuring input
  AbortMeasuringInput := 6000,  
  /// Trigger "Actions" based on I/O related events (e.g. change of DI’s state)
  SetTriggerRegister := 3004,  
  /// Trigger "Actions" based on physical events (e.g. force limit reached)
  SetTriggerLimit := 3002,  
  /// Trigger "Actions" based on physical events (e.g. force limit reached)
  SetTriggerUser := 3005,  
  /// Trigger "Actions" based on incoming error event
  SetTriggerError := 3001,  
  /// "Action" that initiates specified events when triggered
  ReactAtTrigger := 3000,  
  /// Wait to process next command in sequence until trigger signal is received
  WaitForTrigger := 3006,  
  /// Read specific parameter of the robot
  ReadSystemVariable := 5109,  
  /// Change value of specific vendor parameter
  WriteSystemVariable := 5206,  
  /// Calculate Forward Kinematic
  CalculateForwardKinematic := 7203,  
  /// Calculate Inverse Kinematic
  CalculateInverseKinematic := 7204,  
  /// Calculate cartesian position from existing cartesian position
  CalculateCartesianPosition := 7200,  
  /// Calculate tool (TCP) with four-point method
  CalculateTool := 7202,  
  /// Calculate frame with three-point method
  CalculateFrame := 7201,  
  /// Cancel currently active move command and continue with the next buffered command
  ActivateNextCommand := 7000,  
  /// Transform a defined position in space
  ShiftPosition := 7205,  
  /// Trigger an action based on a motion-related parameter (e.g. progress of trajectory)
  SetTriggerMotion := 3003,  
  /// Release robot arm’s brakes
  OpenBrake := 7100,  
  /// Call subprogram stored in RC from PLC
  CallSubprogram := 7001,  
  /// Writes cyclic data of called subprogram
  WriteCallSubprogramCyclic := 2, // No function code
  /// Reads cyclic data of called subprogram
  ReadCallSubprogramCyclic := 3, // No function code
  /// Stops an active subprogram
  StopSubprogram := 7008,  
  /// Switch path mode between high and low accuracy
  PathAccuracyMode := 7401,  
  /// Activate/Deactivate functionality to avoid singularities
  AvoidSingularity := 7400,  
  /// Enables the RC to apply user-defined force/torque through RA’s TCP movement
  ForceControl := 7301,  
  /// Commands specified reaction from RA when defined force/torque detected
  ForceLimit := 7302,  
  /// Read actual force/torque at TCP
  ReadActualForce := 5110,  
  /// Activate robot cycle brake test and give feedback to PLC
  BrakeTest := 7101,  
  /// Push robot: Robot calculates opposite vector and moves slowly in that direction
  SoftSwitchTCP := 7300,  
  /// Create spline on RC from positions stored in PLC
  CreateSpline := 2600,  
  /// Delete spline previously created on RC
  DeleteSpline := 2601,  
  /// Move spline previously created on RC
  MoveSpline := 2603,  
  /// Create and move spline on RC simultaneously
  DynamicSpline := 2602,  
  /// Automatic detection of load data
  LoadMeasurementAutomatic := 7006,  
  /// Sequential detection of load data
  LoadMeasurementSequential := 7007,  
  /// Turn on/off the collision detection
  CollisionDetection := 7003,  
  /// Move the robot axes by hand
  FreeDrive := 7002,  
  /// Measure the length of objects in the cartesian space, execution time for specified section of a job or signal output time of a specified signal
  UnitMeasurement := 7004   
)UINT;
END_TYPE

// Library/Enumerations/Type/ConveyorType
{attribute 'qualified_only'}
// ------------------------------------------------------------------------- 
//  SRCI Robot Library                                                
// ------------------------------------------------------------------------- 
//                                                                           
//  Object:      ConveyorType                                       
//  Author:      Thorsten Brach                                                
//  Date:        2024-06-01
//
//  Description:                                              
//   
//                                                                           
//  Copyright: 
//    (C) 2024 Thorsten Brach. All rights reserved                                                                                                                                            
//             Licensed under the LGPL-3.0 license.
//                                                                           
//  Disclaimer:                                                                           
//    This project is provided without any guarantee and can be used for   
//    private and commercial purposes. Any use is at the user’s 
//    own risk and responsibility.
//
// -------------------------------------------------------------------------
TYPE ConveyorType :
(
  /// Linear Conveyor Tracking (default)
  LINEAR_CONVEYOR_TRACKING := 0,
  /// Circular Conveyor Tracking
  CIRCULAR_CONVEYOR_TRACKING := 1
)USINT;
END_TYPE

// Library/Enumerations/Type/MessageType
{attribute 'qualified_only'}
// ------------------------------------------------------------------------- 
//  SRCI Robot Library                                                
// ------------------------------------------------------------------------- 
//                                                                           
//  Object:      MessageType                                       
//  Author:      Thorsten Brach                                                
//  Date:        2024-06-01
//
//  Description:                                              
//   
//                                                                           
//  Copyright: 
//    (C) 2024 Thorsten Brach. All rights reserved                                                                                                                                            
//             Licensed under the LGPL-3.0 license.
//                                                                           
//  Disclaimer:                                                                           
//    This project is provided without any guarantee and can be used for   
//    private and commercial purposes. Any use is at the user’s 
//    own risk and responsibility.
//
// -------------------------------------------------------------------------
TYPE MessageType :
(
  /// RI related messages
  RI := 1,
  /// RC related messages
  RC := 2,
  /// RA related messages
  RA := 3, 
  /// Command related messages
  CMD := 4 
)USINT;
END_TYPE

// Library/Enumerations/Type/ReferenceType
{attribute 'qualified_only'}
// ------------------------------------------------------------------------- 
//  SRCI Robot Library                                                
// ------------------------------------------------------------------------- 
//                                                                           
//  Object:      ReferenceType                                       
//  Author:      Thorsten Brach                                                
//  Date:        2024-06-01
//
//  Description:                                              
//   
//                                                                           
//  Copyright: 
//    (C) 2024 Thorsten Brach. All rights reserved                                                                                                                                            
//             Licensed under the LGPL-3.0 license.
//                                                                           
//  Disclaimer:                                                                           
//    This project is provided without any guarantee and can be used for   
//    private and commercial purposes. Any use is at the user’s 
//    own risk and responsibility.
//
// -------------------------------------------------------------------------
TYPE ReferenceType :
(
  /// Distance is applied in the Tool coordinate system. 
  /// The setting of the parameter FrameNo will be ignored.
  TOOL  := 0,
  /// Distance is applied in the Frame coordinate system.
  /// The settings of the ToolNo are also effective and must be considered. 
  FRAME := 1
)USINT;
END_TYPE

// Library/Enumerations/Type/UnitType
{attribute 'qualified_only'}
// ------------------------------------------------------------------------- 
//  SRCI Robot Library                                                
// ------------------------------------------------------------------------- 
//                                                                           
//  Object:      UnitType                                       
//  Author:      Thorsten Brach                                                
//  Date:        2024-06-01
//
//  Description:                                              
//   
//                                                                           
//  Copyright: 
//    (C) 2024 Thorsten Brach. All rights reserved                                                                                                                                            
//             Licensed under the LGPL-3.0 license.
//                                                                           
//  Disclaimer:                                                                           
//    This project is provided without any guarantee and can be used for   
//    private and commercial purposes. Any use is at the user’s 
//    own risk and responsibility.
//
// -------------------------------------------------------------------------
TYPE UnitType :
(
  /// Volt
  VOLT   := 0,
  /// Ampere
  AMPERE := 1
)USINT;
END_TYPE

// Library/POUs/Additional/MC_AbortMeasuringInput/Structures/AbortMeasuringInputOutCmd
{attribute 'pack_mode' := '1'} 
// ------------------------------------------------------------------------- 
//  SRCI Robot Library                                                
// ------------------------------------------------------------------------- 
//                                                                           
//  Object:      AbortMeasuringInputOutCmd                                       
//  Author:      Thorsten Brach                                                
//  Date:        2024-06-21
//
//  Description:                                              
//   
//                                                                           
//  Copyright: 
//    (C) 2024 Thorsten Brach. All rights reserved                                                                                                                                            
//             Licensed under the LGPL-3.0 license.
//                                                                           
//  Disclaimer:                                                                           
//    This project is provided without any guarantee and can be used for   
//    private and commercial purposes. Any use is at the user’s 
//    own risk and responsibility.
//
// -------------------------------------------------------------------------
TYPE AbortMeasuringInputOutCmd :
STRUCT
END_STRUCT
END_TYPE

// Library/POUs/Additional/MC_AbortMeasuringInput/Structures/AbortMeasuringInputParCmd
{attribute 'pack_mode' := '1'} 
// ------------------------------------------------------------------------- 
//  SRCI Robot Library                                                
// ------------------------------------------------------------------------- 
//                                                                           
//  Object:      AbortMeasuringInputParCmd                                       
//  Author:      Thorsten Brach                                                
//  Date:        2024-06-21
//
//  Description:                                              
//   
//                                                                           
//  Copyright: 
//    (C) 2024 Thorsten Brach. All rights reserved                                                                                                                                            
//             Licensed under the LGPL-3.0 license.
//                                                                           
//  Disclaimer:                                                                           
//    This project is provided without any guarantee and can be used for   
//    private and commercial purposes. Any use is at the user’s 
//    own risk and responsibility.
//
// -------------------------------------------------------------------------
TYPE AbortMeasuringInputParCmd :
STRUCT
  /// Define an active measurement that is to be aborted.
  /// •  0: Abort all existing measurement
  /// • >0: Abort the measurement with the specific MeasuringID
  MeasuringID        : UINT;
END_STRUCT
END_TYPE

// Library/POUs/Additional/MC_AbortMeasuringInput/Structures/AbortMeasuringInputRecvData
{attribute 'pack_mode' := '1'} 
// ------------------------------------------------------------------------- 
//  SRCI Robot Library                                                
// ------------------------------------------------------------------------- 
//                                                                           
//  Object:      AbortMeasuringInputRecvData                                       
//  Author:      Thorsten Brach                                                
//  Date:        2024-06-21
//
//  Description:                                              
//   
//                                                                           
//  Copyright: 
//    (C) 2024 Thorsten Brach. All rights reserved                                                                                                                                            
//             Licensed under the LGPL-3.0 license.
//                                                                           
//  Disclaimer:                                                                           
//    This project is provided without any guarantee and can be used for   
//    private and commercial purposes. Any use is at the user’s 
//    own risk and responsibility.
//
// -------------------------------------------------------------------------
TYPE AbortMeasuringInputRecvData EXTENDS RspHeader :
STRUCT
END_STRUCT
END_TYPE

// Library/POUs/Additional/MC_AbortMeasuringInput/Structures/AbortMeasuringInputSendData
{attribute 'pack_mode' := '1'}
// ------------------------------------------------------------------------- 
//  SRCI Robot Library                                                
// ------------------------------------------------------------------------- 
//                                                                           
//  Object:      AbortMeasuringInputSendData                                       
//  Author:      Thorsten Brach                                                
//  Date:        2024-06-21
//
//  Description:                                              
//   
//                                                                           
//  Copyright: 
//    (C) 2024 Thorsten Brach. All rights reserved                                                                                                                                            
//             Licensed under the LGPL-3.0 license.
//                                                                           
//  Disclaimer:                                                                           
//    This project is provided without any guarantee and can be used for   
//    private and commercial purposes. Any use is at the user’s 
//    own risk and responsibility.
//
// -------------------------------------------------------------------------
TYPE AbortMeasuringInputSendData EXTENDS CmdHeader:   
STRUCT
  /// Define an active measurement that is to be aborted.
  /// •  0: Abort all existing measurement
  /// • >0: Abort the measurement with the specific MeasuringID
  MeasuringID        : UINT;
END_STRUCT
END_TYPE

// Library/POUs/Additional/MC_ActivateNextCommand/Structures/ActivateNextCommandOutCmd
{attribute 'pack_mode' := '1'} 
// ------------------------------------------------------------------------- 
//  SRCI Robot Library                                                
// ------------------------------------------------------------------------- 
//                                                                           
//  Object:      ActivateNextCommandOutCmd                                       
//  Author:      Thorsten Brach                                                
//  Date:        2024-06-01
//
//  Description:                                              
//   
//                                                                           
//  Copyright: 
//             Licensed under the LGPL-3.0 license.
//    (C) 2024 Thorsten Brach. All rights reserved                                                                                                                                            
//                                                                           
//  Disclaimer:                                                                           
//    This project is provided without any guarantee and can be used for   
//    private and commercial purposes. Any use is at the user’s 
//    own risk and responsibility.
//
// -------------------------------------------------------------------------
TYPE ActivateNextCommandOutCmd :
STRUCT
  /// Unique system-generated ID of the "Action" when the function is triggered.
  /// • >0: The "Action" is started by the trigger function with identical FollowID.
  /// • <0: The "Action" is stopped by the trigger function with identical FollowID.
  /// For more information see chapter 5.5.12.4 EmitterID, ListenerID, FollowID and OriginID
  OriginID           : INT;
  /// Relates to ListenerID >0
  /// Number of successful trigger -based command invocations
  /// For more information refer to chapter 5.5.12.4.
  InvocationCounter  : USINT;
END_STRUCT
END_TYPE

// Library/POUs/Additional/MC_ActivateNextCommand/Structures/ActivateNextCommandParCmd
{attribute 'pack_mode' := '1'} 
// ------------------------------------------------------------------------- 
//  SRCI Robot Library                                                
// ------------------------------------------------------------------------- 
//                                                                           
//  Object:      ActivateNextCommandParCmd                                       
//  Author:      Thorsten Brach                                                
//  Date:        2024-06-01
//
//  Description:                                              
//   
//                                                                           
//  Copyright: 
//    (C) 2024 Thorsten Brach. All rights reserved                                                                                                                                            
//             Licensed under the LGPL-3.0 license.
//                                                                           
//  Disclaimer:                                                                           
//    This project is provided without any guarantee and can be used for   
//    private and commercial purposes. Any use is at the user’s 
//    own risk and responsibility.
//
// -------------------------------------------------------------------------
TYPE ActivateNextCommandParCmd :
STRUCT
  /// Processing mode
  ProcessingMode : ProcessingMode;
  /// ID of the trigger function that may be triggered:
  /// • 0: Immediately (default). - Start executing THIS function immediately.
  /// • >0: Triggero Start executing when the trigger function with the identical EmitterID is called.
  /// For more information see chapter 5.5.12.4.
  ListenerID     : SINT;
END_STRUCT
END_TYPE

